// TIA Portal V18 export
DATA_BLOCK "LED_lampTestAtStartup_DB"   // DB8
VERSION : 0.1
// stored: AutoNumber true, DBAccessibleFromOPCUA true, InstanceOfName LED_lampTestAtStartup, InstanceOfType FB
"LED_lampTestAtStartup"
   // VAR_IN_OUT
   //    HMI_TEST_ALL_LEDS : Bool;
   // END_VAR
   // VAR
   //    IEC_Timer_0_Instance { S7_SetPoint := 'True'} : TON_TIME;
   //    mem : Bool;
   // END_VAR
BEGIN
END_DATA_BLOCK
